(* PLC project Unnamed, Unknown Unnamed 1 *)
(* stored: creationDateTime 2026-05-08T16:57:58, modificationDateTime 2026-05-08T16:57:58 *)

FUNCTION_BLOCK Decoder7Seg
  VAR_INPUT
    InputTal : INT;
  END_VAR
  VAR_OUTPUT
    a : BOOL;
    b : BOOL;
    c : BOOL;
    d : BOOL;
    e : BOOL;
    f : BOOL;
    g : BOOL;
  END_VAR

            CASE InputTal OF
    0, 10: a:=1; b:=1; c:=1; d:=1; e:=1; f:=1; g:=0;
    1: a:=0; b:=1; c:=1; d:=0; e:=0; f:=0; g:=0;
    2: a:=1; b:=1; c:=0; d:=1; e:=1; f:=0; g:=1;
    3: a:=1; b:=1; c:=1; d:=1; e:=0; f:=0; g:=1;
    4: a:=0; b:=1; c:=1; d:=0; e:=0; f:=1; g:=1;
    5: a:=1; b:=0; c:=1; d:=1; e:=0; f:=1; g:=1;
    6: a:=1; b:=0; c:=1; d:=1; e:=1; f:=1; g:=1;
    7: a:=1; b:=1; c:=1; d:=0; e:=0; f:=0; g:=0;
    8: a:=1; b:=1; c:=1; d:=1; e:=1; f:=1; g:=1;
    9: a:=1; b:=1; c:=1; d:=1; e:=0; f:=1; g:=1;
    ELSE
       a:=0; b:=0; c:=0; d:=0; e:=0; f:=0; g:=0;
END_CASE;
          
END_FUNCTION_BLOCK

PROGRAM main
  VAR
    seg_a AT %QX0.0 : BOOL;
    seg_b AT %QX0.1 : BOOL;
    seg_c AT %QX0.2 : BOOL;
    seg_d AT %QX0.3 : BOOL;
    seg_e AT %QX0.4 : BOOL;
    seg_f AT %QX0.5 : BOOL;
    seg_g AT %QX0.6 : BOOL;
    BtnGreen AT %IX0.0 : BOOL;
  END_VAR
  VAR
    counter : INT;
    seg1_display : Decoder7Seg;
    resetValue : INT := 9;
    presetValue : INT := 10;
    resetTrigger : BOOL;
    CTU1 : CTU;
    TON0 : TON;
    TON_Timer : TIME := T#30ms;
    TON_trigger : BOOL;
    Seg1_trigger : BOOL;
  END_VAR

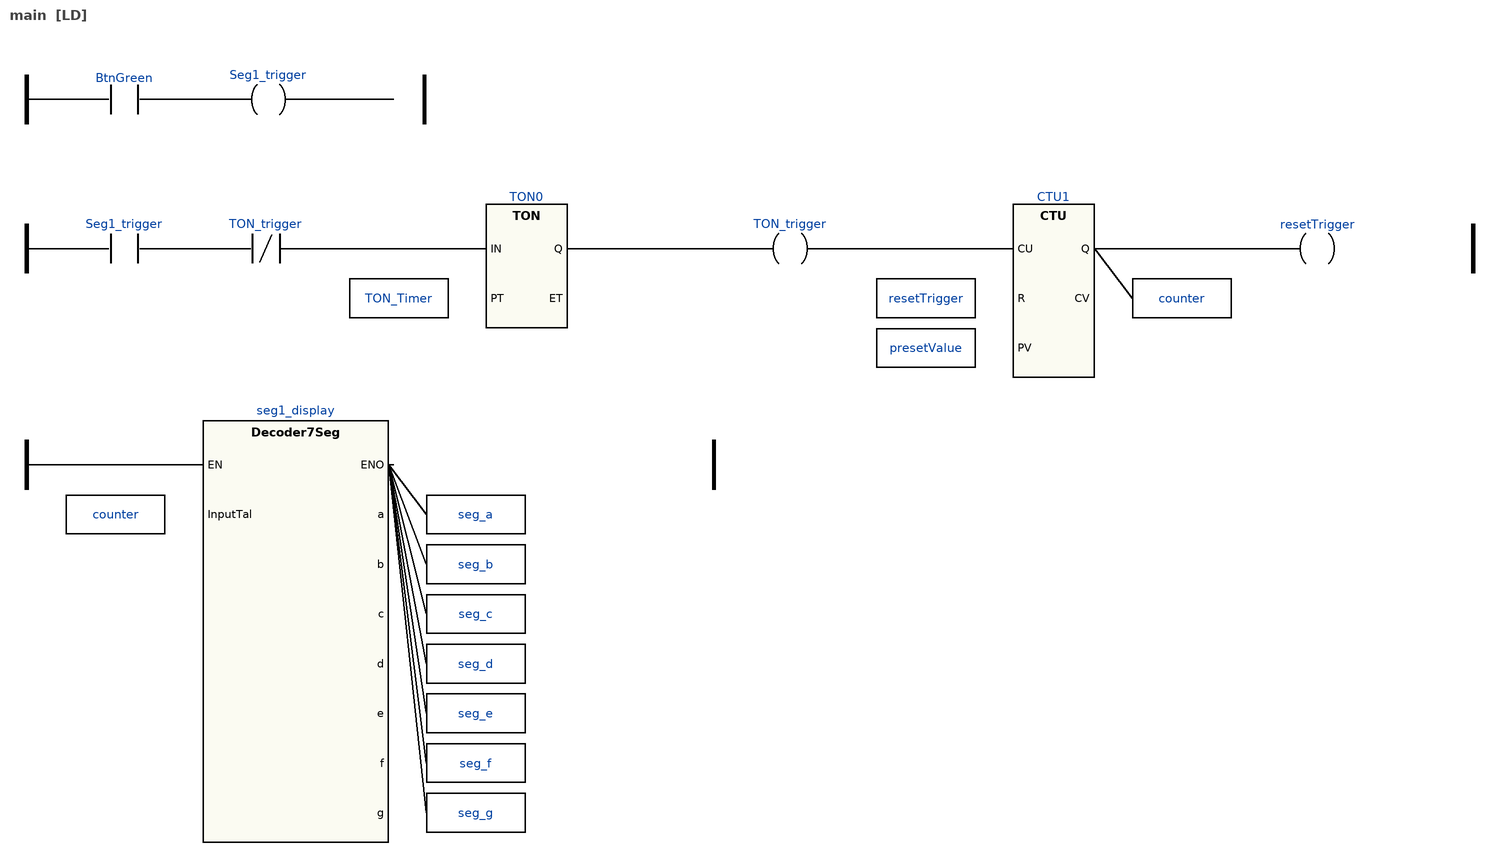
(* LD diagram, written out as Structured Text *)
Seg1_trigger := BtnGreen;
TON0(IN := Seg1_trigger AND NOT TON_trigger, PT := TON_Timer);
TON_trigger := TON0.Q;
CTU1(CU := TON0.Q, R := resetTrigger, PV := presetValue);
resetTrigger := CTU1.Q;
counter := CTU1.CV;
seg1_display(InputTal := counter);
seg_a := seg1_display.a;
seg_b := seg1_display.b;
seg_c := seg1_display.c;
seg_d := seg1_display.d;
seg_e := seg1_display.e;
seg_f := seg1_display.f;
seg_g := seg1_display.g;
END_PROGRAM

CONFIGURATION Config0
  RESOURCE Res0 ON PLC
    TASK task0(INTERVAL := T#20ms, PRIORITY := 1);
    PROGRAM instance0 WITH task0 : main;
  END_RESOURCE
END_CONFIGURATION
